FUNCTION_BLOCK ConveyorMain
VAR_INPUT
    Start       : BOOL;
    Stop        : BOOL;
    FaultReset  : BOOL;
END_VAR
VAR_OUTPUT
    Running     : BOOL;
    Faulted     : BOOL;
END_VAR
VAR
    RunningInternal : BOOL;
END_VAR


IF FaultReset THEN
    Faulted := FALSE;
END_IF

IF Start AND NOT Faulted THEN
    RunningInternal := TRUE;
END_IF

IF Stop THEN
    RunningInternal := FALSE;
END_IF

Running := RunningInternal;

END_FUNCTION_BLOCK

(* stored: Version 1.1.0.1, ProductVersion 3.1.4026.18
   POU ConveyorMain: Id {62485d5d-0862-4ae4-b31a-2f3308341a09}, SpecialFunc None *)
